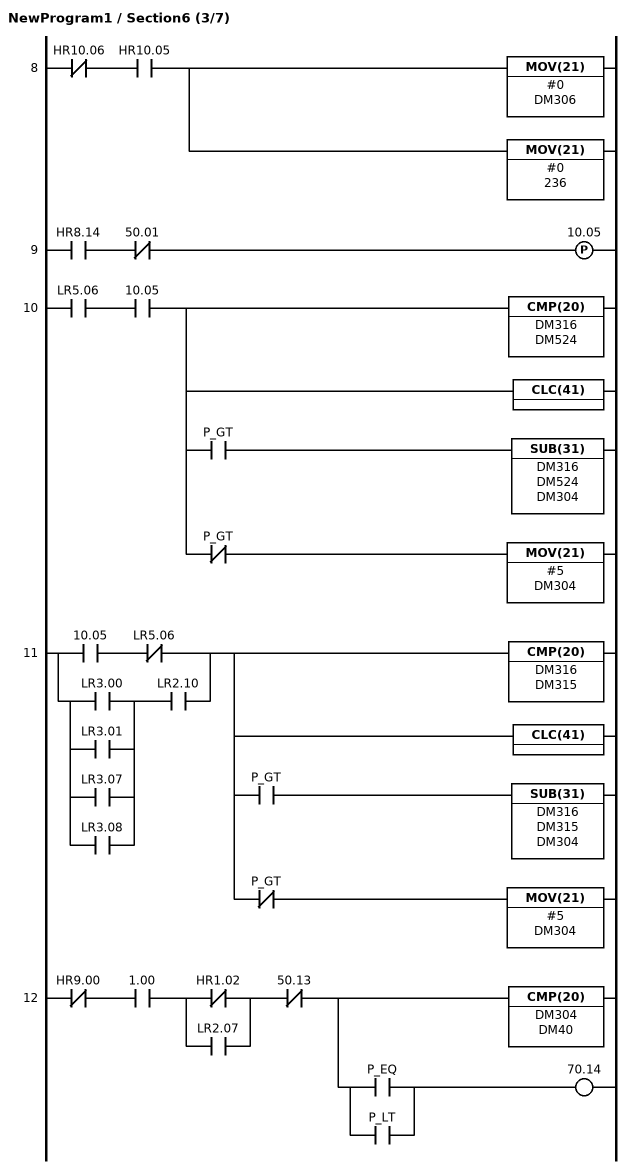
; [picture p48: NewProgram1 / Section6, rungs 8-12]
; rung 8
LDNOT HR10.06
AND HR10.05
MOV(21) #0 DM306
MOV(21) #0 236
; rung 9
LD HR8.14
ANDNOT 50.01
DIFU(13) 10.05
; rung 10
LD LR5.06
AND 10.05
OUT TR0
CMP(20) DM316 DM524
CLC(41)
AND P_GT
SUB(31) DM316 DM524 DM304
LD TR0
ANDNOT P_GT
MOV(21) #5 DM304
; rung 11
LD 10.05
ANDNOT LR5.06
LD LR3.00
OR LR3.01
OR LR3.07
OR LR3.08
AND LR2.10
ORLD
OUT TR0
CMP(20) DM316 DM315
CLC(41)
AND P_GT
SUB(31) DM316 DM315 DM304
LD TR0
ANDNOT P_GT
MOV(21) #5 DM304
; rung 12
LDNOT HR9.00
AND 1.00
LDNOT HR1.02
OR LR2.07
ANDLD
ANDNOT 50.13
CMP(20) DM304 DM40
LD P_EQ
OR P_LT
ANDLD
OUT 70.14

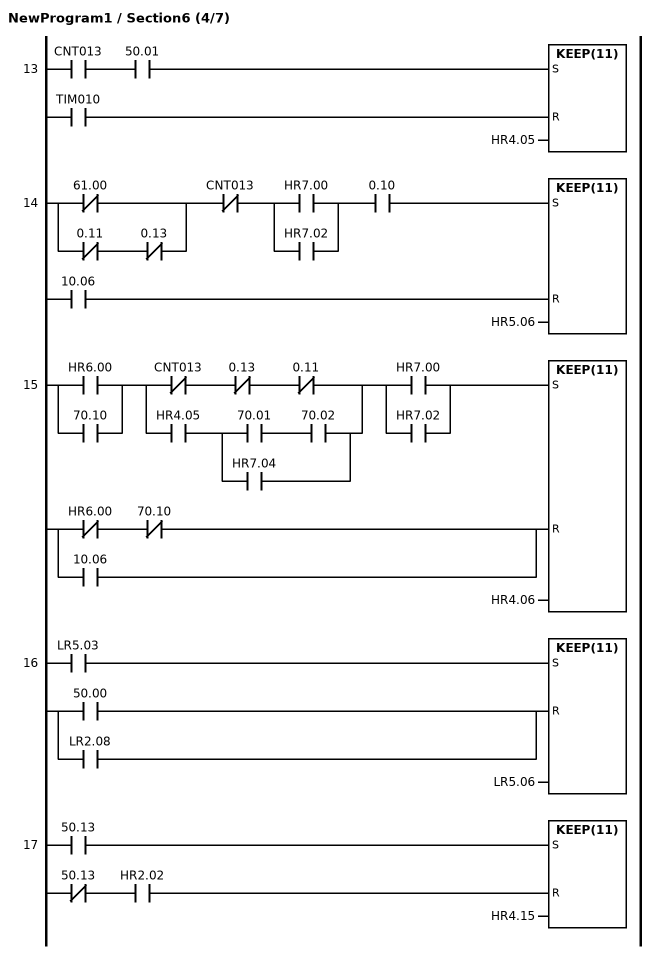
; rung 13
LD CNT013
AND 50.01
LD TIM010
KEEP(11) HR4.05
; rung 14
LDNOT 61.00
LDNOT 0.11
ANDNOT 0.13
ORLD
ANDNOT CNT013
LD HR7.00
OR HR7.02
ANDLD
AND 0.10
LD 10.06
KEEP(11) HR5.06
; rung 15
LD HR6.00
OR 70.10
LDNOT CNT013
ANDNOT 0.13
ANDNOT 0.11
LD HR4.05
LD 70.01
AND 70.02
OR HR7.04
ANDLD
ORLD
ANDLD
LD HR7.00
OR HR7.02
ANDLD
LDNOT HR6.00
ANDNOT 70.10
OR 10.06
KEEP(11) HR4.06
; rung 16
LD LR5.03
LD 50.00
OR LR2.08
KEEP(11) LR5.06
; rung 17
LD 50.13
LDNOT 50.13
AND HR2.02
KEEP(11) HR4.15

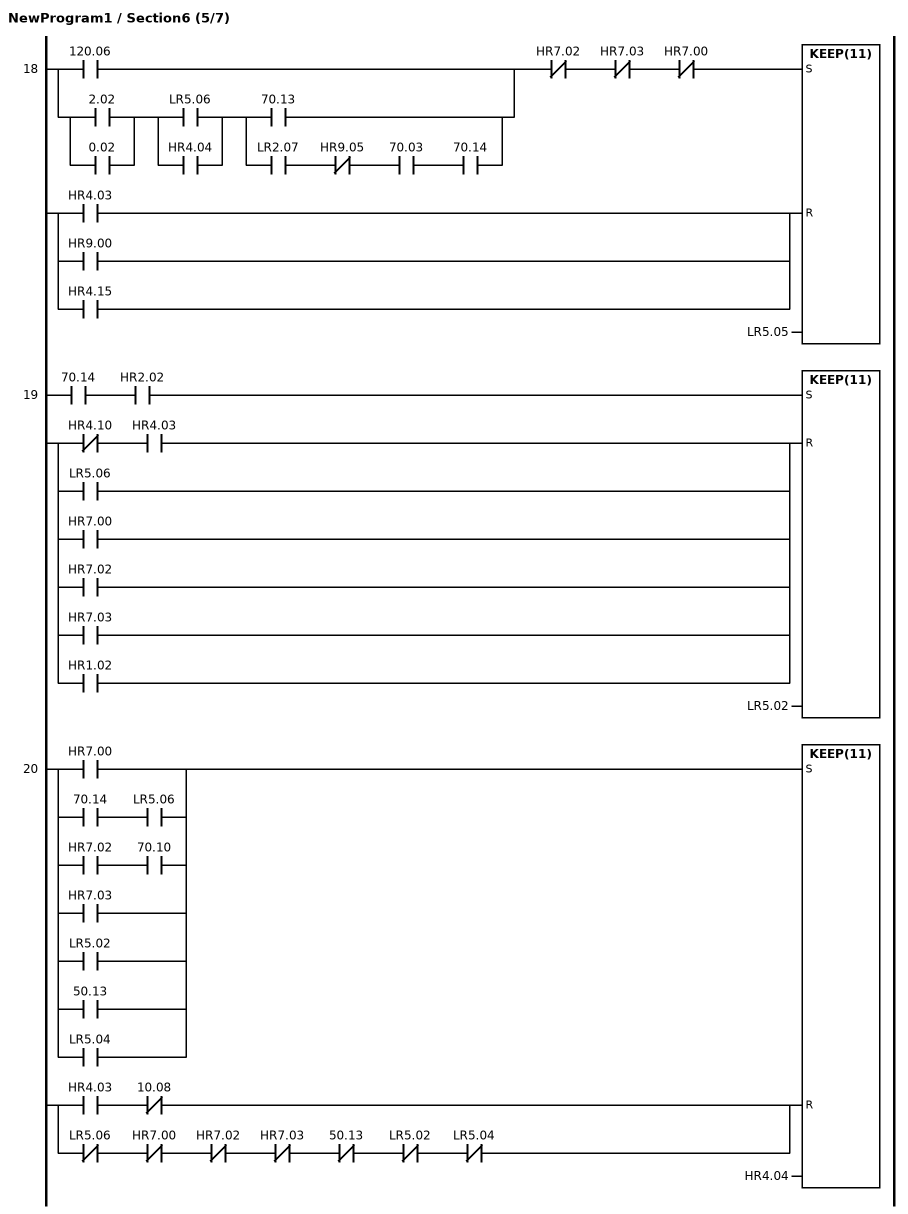
; rung 18
LD 120.06
LD 2.02
OR 0.02
LD LR5.06
OR HR4.04
ANDLD
LD 70.13
LD LR2.07
ANDNOT HR9.05
AND 70.03
AND 70.14
ORLD
ANDLD
ORLD
ANDNOT HR7.02
ANDNOT HR7.03
ANDNOT HR7.00
LD HR4.03
OR HR9.00
OR HR4.15
KEEP(11) LR5.05
; rung 19
LD 70.14
AND HR2.02
LDNOT HR4.10
AND HR4.03
OR LR5.06
OR HR7.00
OR HR7.02
OR HR7.03
OR HR1.02
KEEP(11) LR5.02
; rung 20
LD HR7.00
LD 70.14
AND LR5.06
ORLD
LD HR7.02
AND 70.10
ORLD
OR HR7.03
OR LR5.02
OR 50.13
OR LR5.04
LD HR4.03
ANDNOT 10.08
LDNOT LR5.06
ANDNOT HR7.00
ANDNOT HR7.02
ANDNOT HR7.03
ANDNOT 50.13
ANDNOT LR5.02
ANDNOT LR5.04
ORLD
KEEP(11) HR4.04

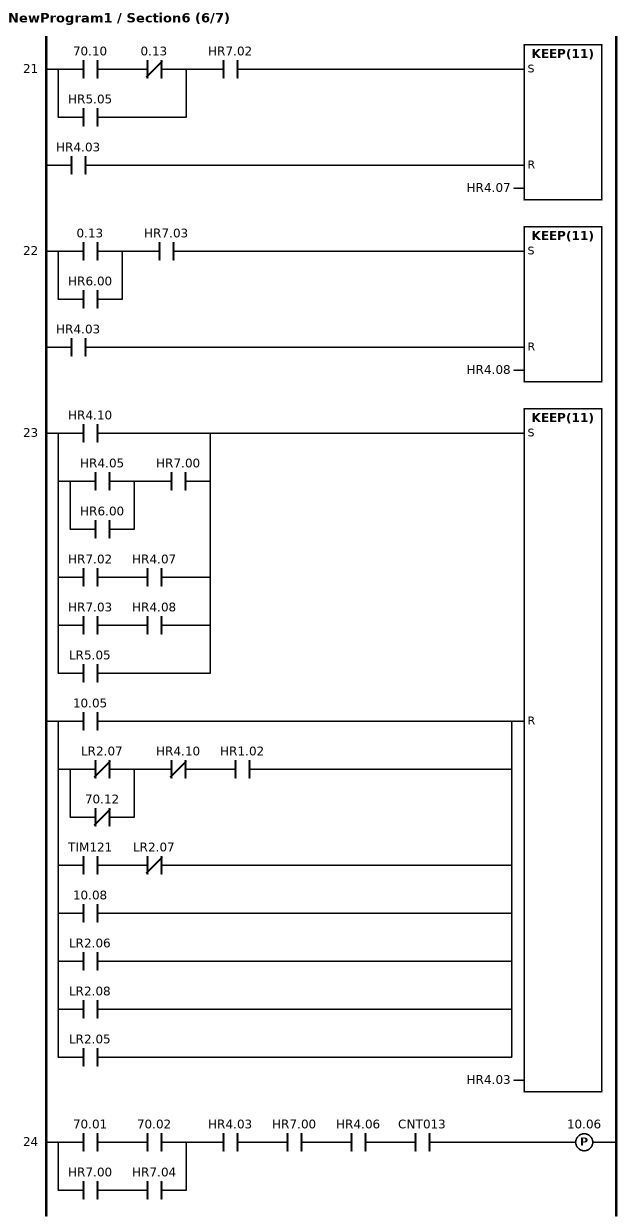
; rung 21
LD 70.10
ANDNOT 0.13
OR HR5.05
AND HR7.02
LD HR4.03
KEEP(11) HR4.07
; rung 22
LD 0.13
OR HR6.00
AND HR7.03
LD HR4.03
KEEP(11) HR4.08
; rung 23
LD HR4.10
LD HR4.05
OR HR6.00
AND HR7.00
ORLD
LD HR7.02
AND HR4.07
ORLD
LD HR7.03
AND HR4.08
ORLD
OR LR5.05
LD 10.05
LDNOT LR2.07
ORNOT 70.12
ANDNOT HR4.10
AND HR1.02
ORLD
LD TIM121
ANDNOT LR2.07
ORLD
OR 10.08
OR LR2.06
OR LR2.08
OR LR2.05
KEEP(11) HR4.03
; rung 24
LD 70.01
AND 70.02
LD HR7.00
AND HR7.04
ORLD
AND HR4.03
AND HR7.00
AND HR4.06
AND CNT013
DIFU(13) 10.06

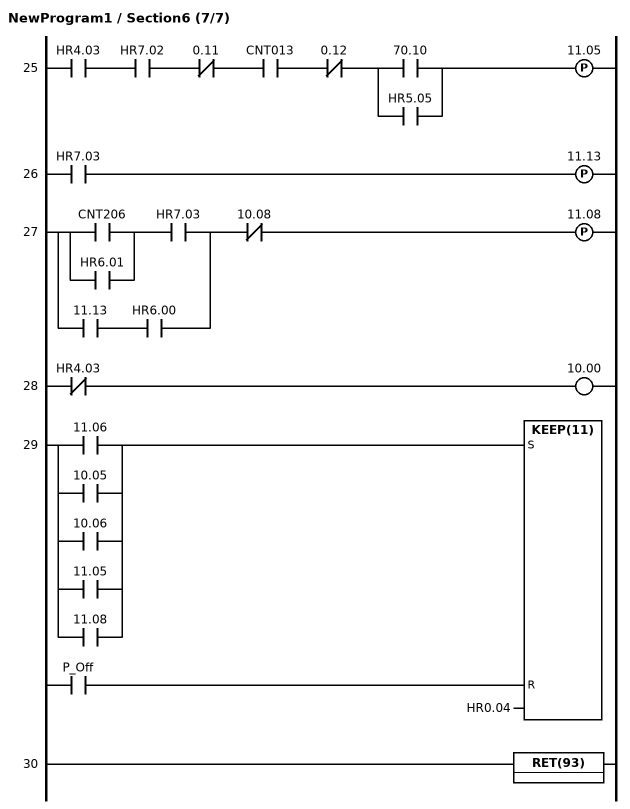
; rung 25
LD HR4.03
AND HR7.02
ANDNOT 0.11
AND CNT013
ANDNOT 0.12
LD 70.10
OR HR5.05
ANDLD
DIFU(13) 11.05
; rung 26
LD HR7.03
DIFU(13) 11.13
; rung 27
LD CNT206
OR HR6.01
AND HR7.03
LD 11.13
AND HR6.00
ORLD
ANDNOT 10.08
DIFU(13) 11.08
; rung 28
LDNOT HR4.03
OUT 10.00
; rung 29
LD 11.06
OR 10.05
OR 10.06
OR 11.05
OR 11.08
LD P_Off
KEEP(11) HR0.04
; rung 30
RET(93)

### Section Section7

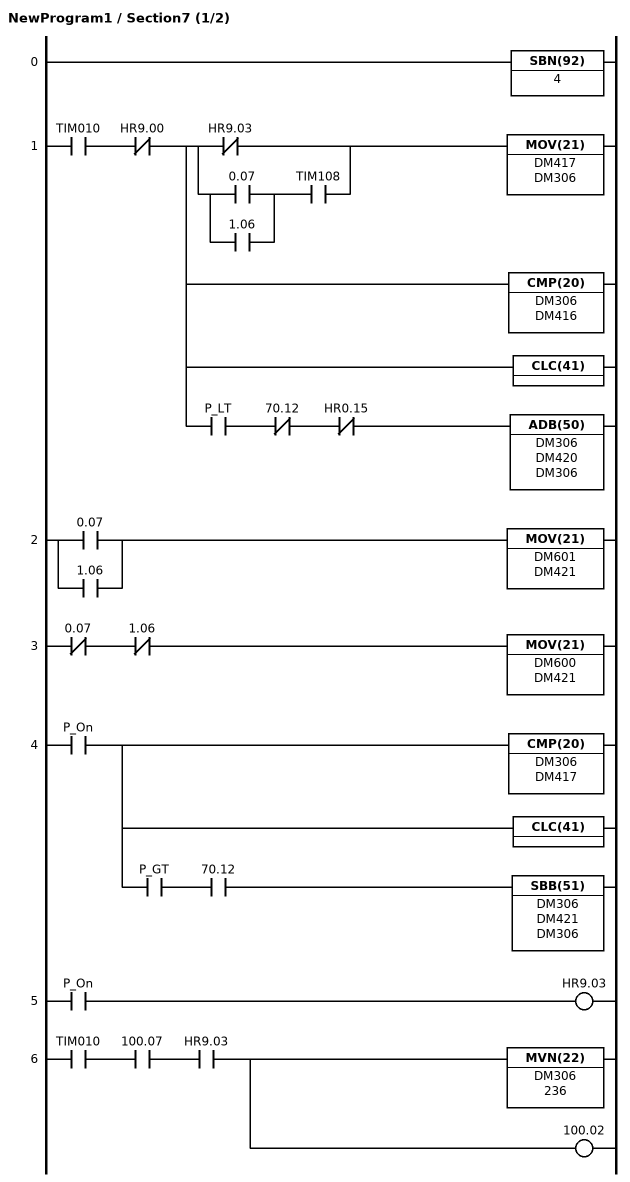
; rung 0
SBN(92) 4
; rung 1
LD TIM010
ANDNOT HR9.00
OUT TR0
LDNOT HR9.03
LD 0.07
OR 1.06
AND TIM108
ORLD
ANDLD
MOV(21) DM417 DM306
LD TR0
CMP(20) DM306 DM416
CLC(41)
AND P_LT
ANDNOT 70.12
ANDNOT HR0.15
ADB(50) DM306 DM420 DM306
; rung 2
LD 0.07
OR 1.06
MOV(21) DM601 DM421
; rung 3
LDNOT 0.07
ANDNOT 1.06
MOV(21) DM600 DM421
; rung 4
LD P_On
CMP(20) DM306 DM417
CLC(41)
AND P_GT
AND 70.12
SBB(51) DM306 DM421 DM306
; rung 5
LD P_On
OUT HR9.03
; rung 6
LD TIM010
AND 100.07
AND HR9.03
MVN(22) DM306 236
OUT 100.02

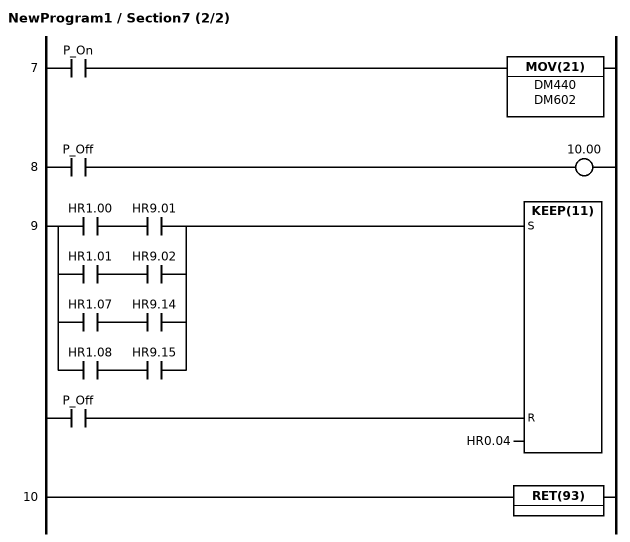
; rung 7
LD P_On
MOV(21) DM440 DM602
; rung 8
LD P_Off
OUT 10.00
; rung 9
LD HR1.00
AND HR9.01
LD HR1.01
AND HR9.02
ORLD
LD HR1.07
AND HR9.14
ORLD
LD HR1.08
AND HR9.15
ORLD
LD P_Off
KEEP(11) HR0.04
; rung 10
RET(93)

### Section Section8

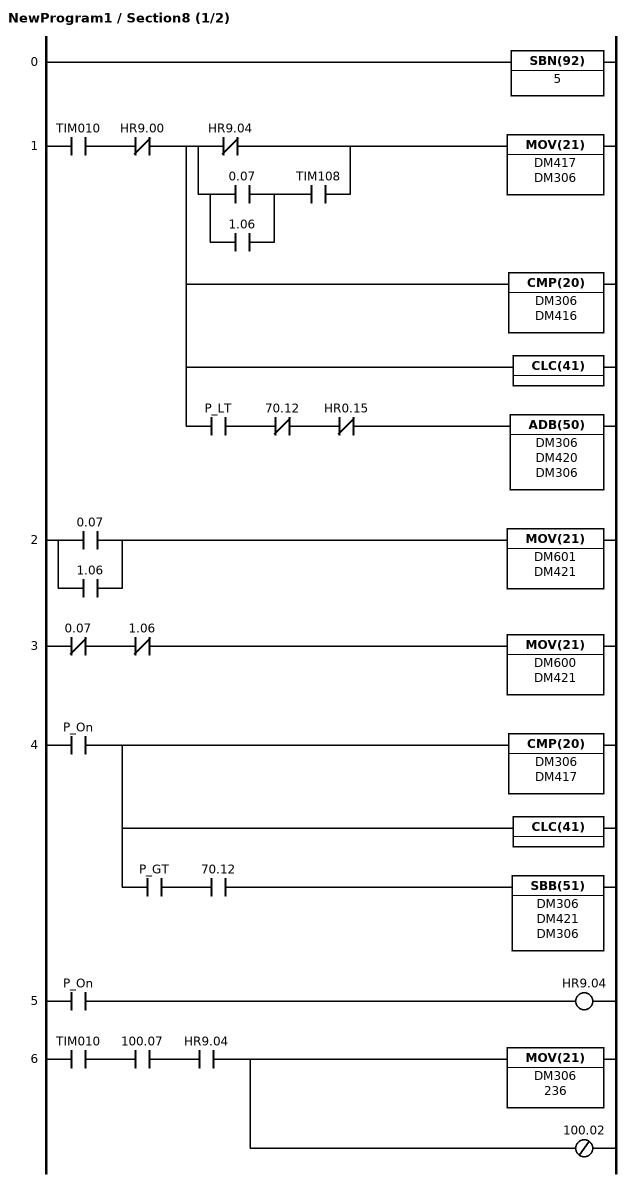
; rung 0
SBN(92) 5
; rung 1
LD TIM010
ANDNOT HR9.00
OUT TR0
LDNOT HR9.04
LD 0.07
OR 1.06
AND TIM108
ORLD
ANDLD
MOV(21) DM417 DM306
LD TR0
CMP(20) DM306 DM416
CLC(41)
AND P_LT
ANDNOT 70.12
ANDNOT HR0.15
ADB(50) DM306 DM420 DM306
; rung 2
LD 0.07
OR 1.06
MOV(21) DM601 DM421
; rung 3
LDNOT 0.07
ANDNOT 1.06
MOV(21) DM600 DM421
; rung 4
LD P_On
CMP(20) DM306 DM417
CLC(41)
AND P_GT
AND 70.12
SBB(51) DM306 DM421 DM306
; rung 5
LD P_On
OUT HR9.04
; rung 6
LD TIM010
AND 100.07
AND HR9.04
MOV(21) DM306 236
OUTNOT 100.02

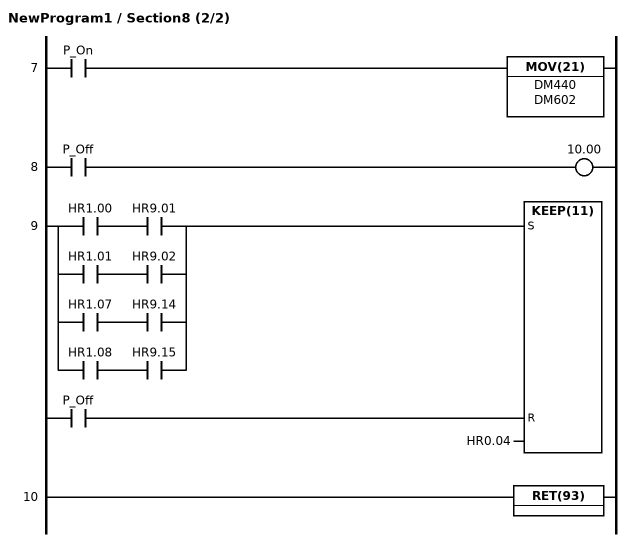
; rung 7
LD P_On
MOV(21) DM440 DM602
; rung 8
LD P_Off
OUT 10.00
; rung 9
LD HR1.00
AND HR9.01
LD HR1.01
AND HR9.02
ORLD
LD HR1.07
AND HR9.14
ORLD
LD HR1.08
AND HR9.15
ORLD
LD P_Off
KEEP(11) HR0.04
; rung 10
RET(93)

### Section Section9

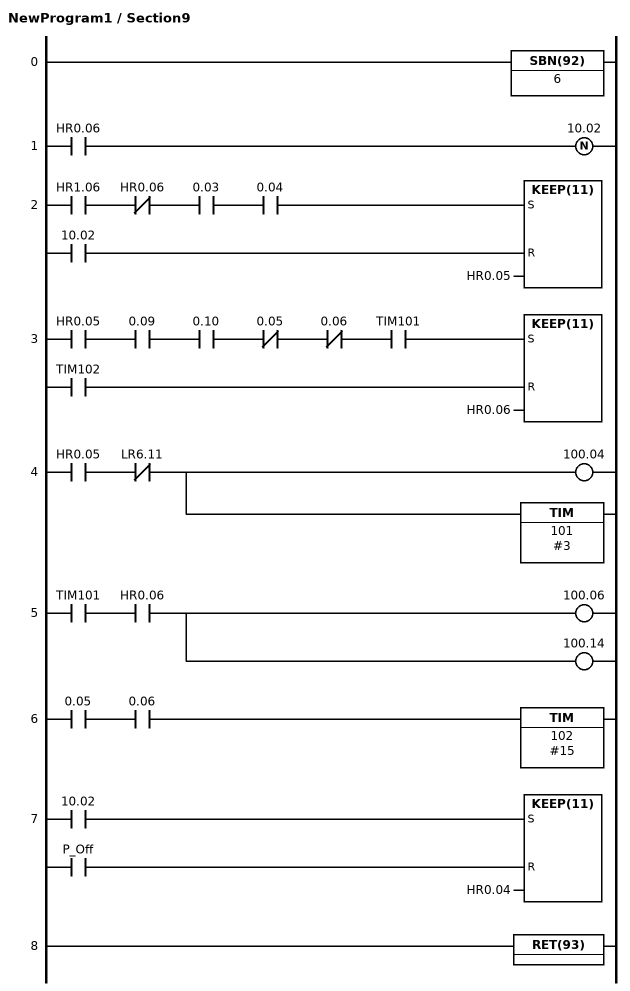
; rung 0
SBN(92) 6
; rung 1
LD HR0.06
DIFD(14) 10.02
; rung 2
LD HR1.06
ANDNOT HR0.06
AND 0.03
AND 0.04
LD 10.02
KEEP(11) HR0.05
; rung 3
LD HR0.05
AND 0.09
AND 0.10
ANDNOT 0.05
ANDNOT 0.06
AND TIM101
LD TIM102
KEEP(11) HR0.06
; rung 4
LD HR0.05
ANDNOT LR6.11
OUT 100.04
TIM 101 #3
; rung 5
LD TIM101
AND HR0.06
OUT 100.06
OUT 100.14
; rung 6
LD 0.05
AND 0.06
TIM 102 #15
; rung 7
LD 10.02
LD P_Off
KEEP(11) HR0.04
; rung 8
RET(93)

### Section Section10

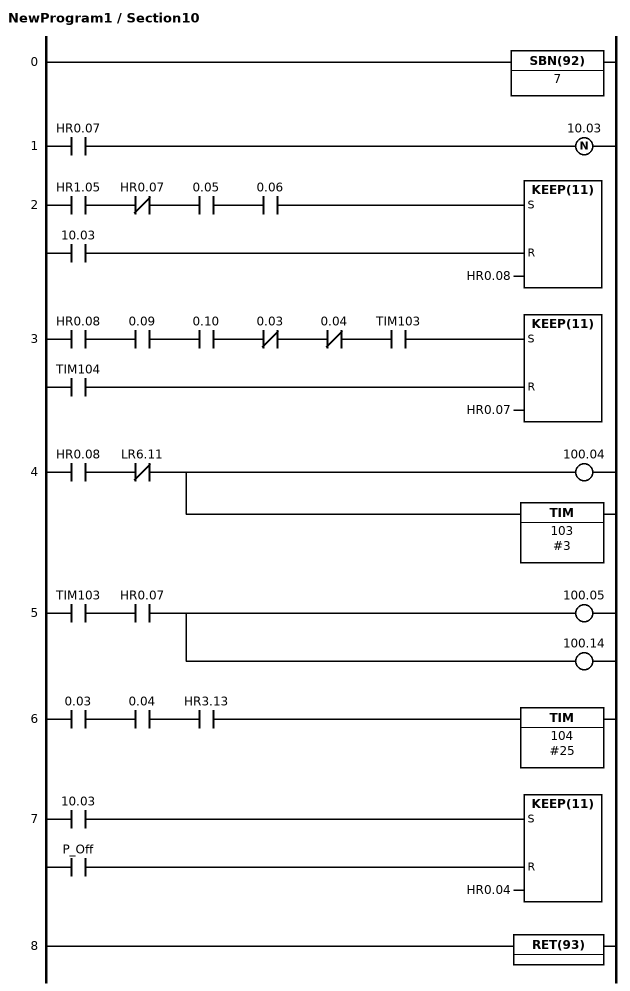
; rung 0
SBN(92) 7
; rung 1
LD HR0.07
DIFD(14) 10.03
; rung 2
LD HR1.05
ANDNOT HR0.07
AND 0.05
AND 0.06
LD 10.03
KEEP(11) HR0.08
; rung 3
LD HR0.08
AND 0.09
AND 0.10
ANDNOT 0.03
ANDNOT 0.04
AND TIM103
LD TIM104
KEEP(11) HR0.07
; rung 4
LD HR0.08
ANDNOT LR6.11
OUT 100.04
TIM 103 #3
; rung 5
LD TIM103
AND HR0.07
OUT 100.05
OUT 100.14
; rung 6
LD 0.03
AND 0.04
AND HR3.13
TIM 104 #25
; rung 7
LD 10.03
LD P_Off
KEEP(11) HR0.04
; rung 8
RET(93)

### Section Section11

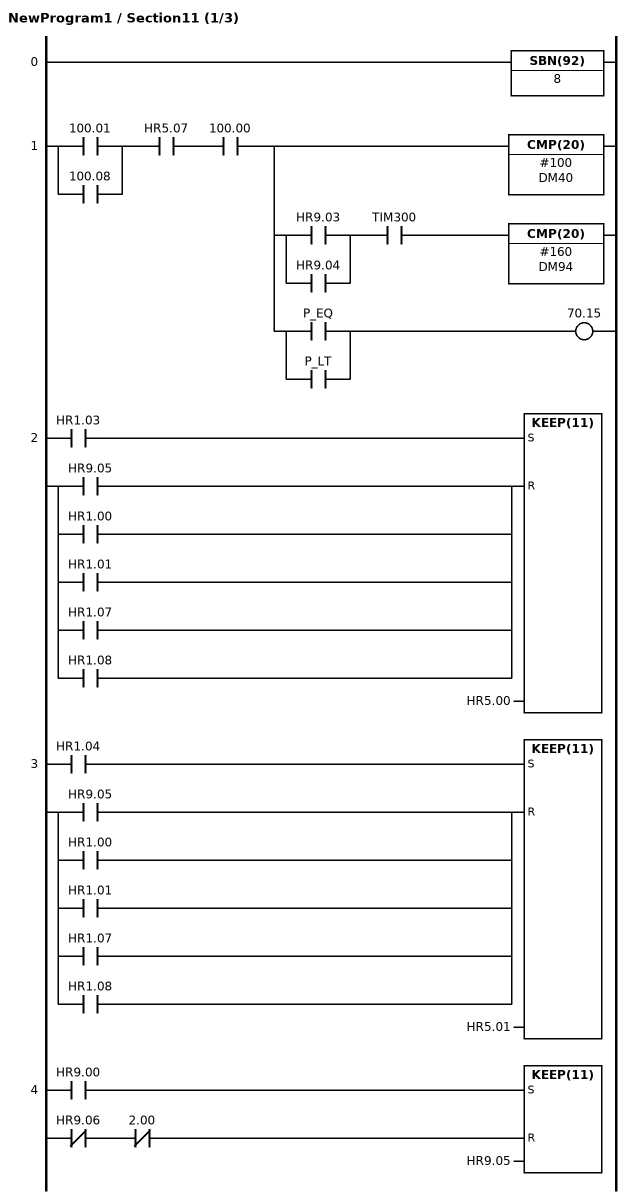
; rung 0
SBN(92) 8
; rung 1
LD 100.01
OR 100.08
AND HR5.07
AND 100.00
OUT TR0
CMP(20) #100 DM40
LD HR9.03
OR HR9.04
ANDLD
AND TIM300
CMP(20) #160 DM94
LD TR0
LD P_EQ
OR P_LT
ANDLD
OUT 70.15
; rung 2
LD HR1.03
LD HR9.05
OR HR1.00
OR HR1.01
OR HR1.07
OR HR1.08
KEEP(11) HR5.00
; rung 3
LD HR1.04
LD HR9.05
OR HR1.00
OR HR1.01
OR HR1.07
OR HR1.08
KEEP(11) HR5.01
; rung 4
LD HR9.00
LDNOT HR9.06
ANDNOT 2.00
KEEP(11) HR9.05

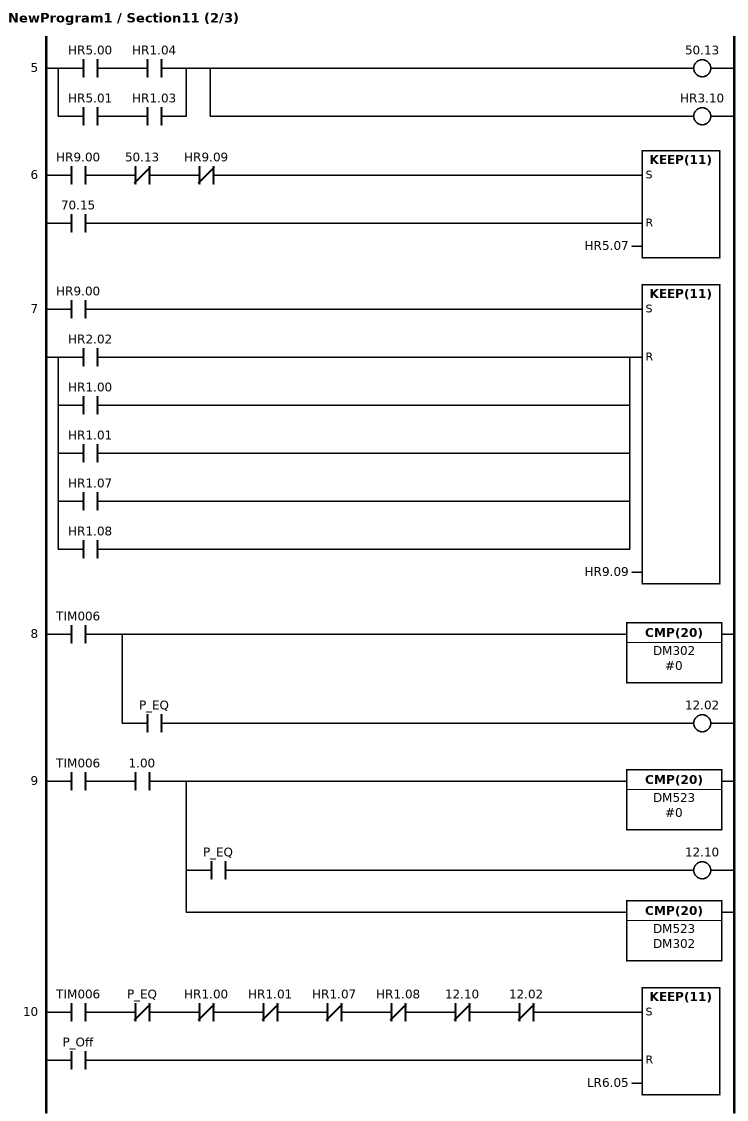
; rung 5
LD HR5.00
AND HR1.04
LD HR5.01
AND HR1.03
ORLD
OUT 50.13
OUT HR3.10
; rung 6
LD HR9.00
ANDNOT 50.13
ANDNOT HR9.09
LD 70.15
KEEP(11) HR5.07
; rung 7
LD HR9.00
LD HR2.02
OR HR1.00
OR HR1.01
OR HR1.07
OR HR1.08
KEEP(11) HR9.09
; rung 8
LD TIM006
CMP(20) DM302 #0
AND P_EQ
OUT 12.02
; rung 9
LD TIM006
AND 1.00
OUT TR0
CMP(20) DM523 #0
AND P_EQ
OUT 12.10
LD TR0
CMP(20) DM523 DM302
; rung 10
LD TIM006
ANDNOT P_EQ
ANDNOT HR1.00
ANDNOT HR1.01
ANDNOT HR1.07
ANDNOT HR1.08
ANDNOT 12.10
ANDNOT 12.02
LD P_Off
KEEP(11) LR6.05

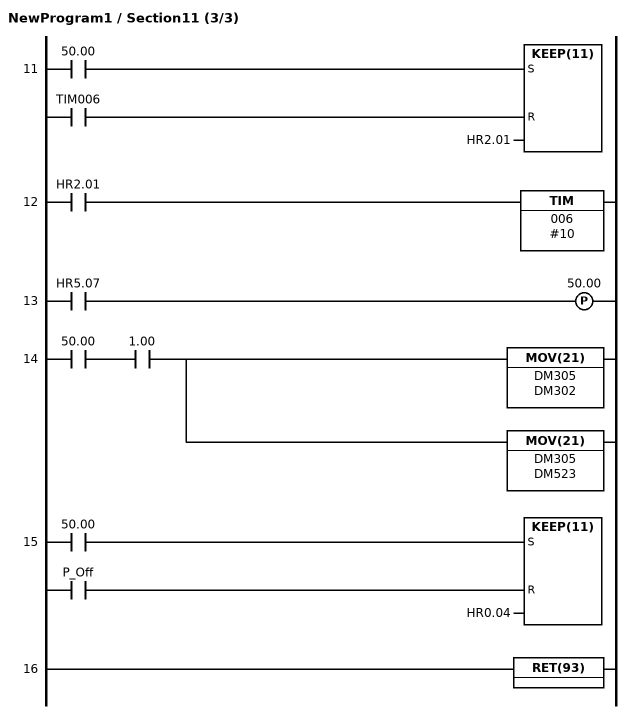
; rung 11
LD 50.00
LD TIM006
KEEP(11) HR2.01
; rung 12
LD HR2.01
TIM 006 #10
; rung 13
LD HR5.07
DIFU(13) 50.00
; rung 14
LD 50.00
AND 1.00
MOV(21) DM305 DM302
MOV(21) DM305 DM523
; rung 15
LD 50.00
LD P_Off
KEEP(11) HR0.04
; rung 16
RET(93)

### Section Section12

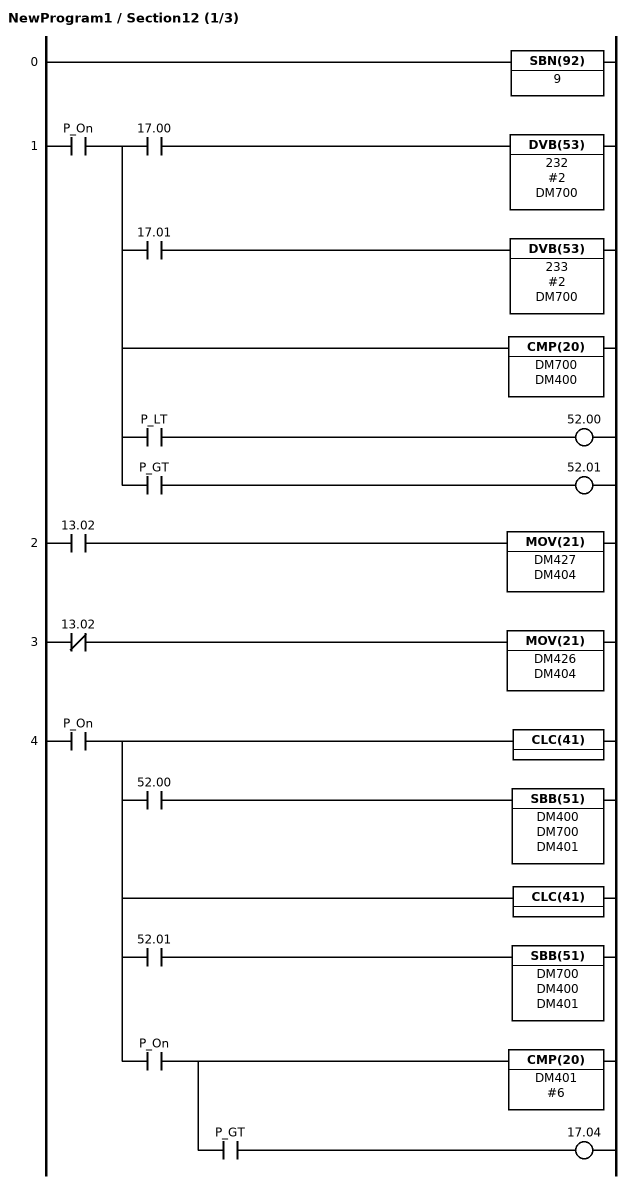
; rung 0
SBN(92) 9
; rung 1
LD P_On
OUT TR0
AND 17.00
DVB(53) 232 #2 DM700
LD TR0
AND 17.01
DVB(53) 233 #2 DM700
LD TR0
CMP(20) DM700 DM400
AND P_LT
OUT 52.00
LD TR0
AND P_GT
OUT 52.01
; rung 2
LD 13.02
MOV(21) DM427 DM404
; rung 3
LDNOT 13.02
MOV(21) DM426 DM404
; rung 4
LD P_On
OUT TR0
CLC(41)
AND 52.00
SBB(51) DM400 DM700 DM401
LD TR0
CLC(41)
AND 52.01
SBB(51) DM700 DM400 DM401
LD TR0
AND P_On
CMP(20) DM401 #6
AND P_GT
OUT 17.04

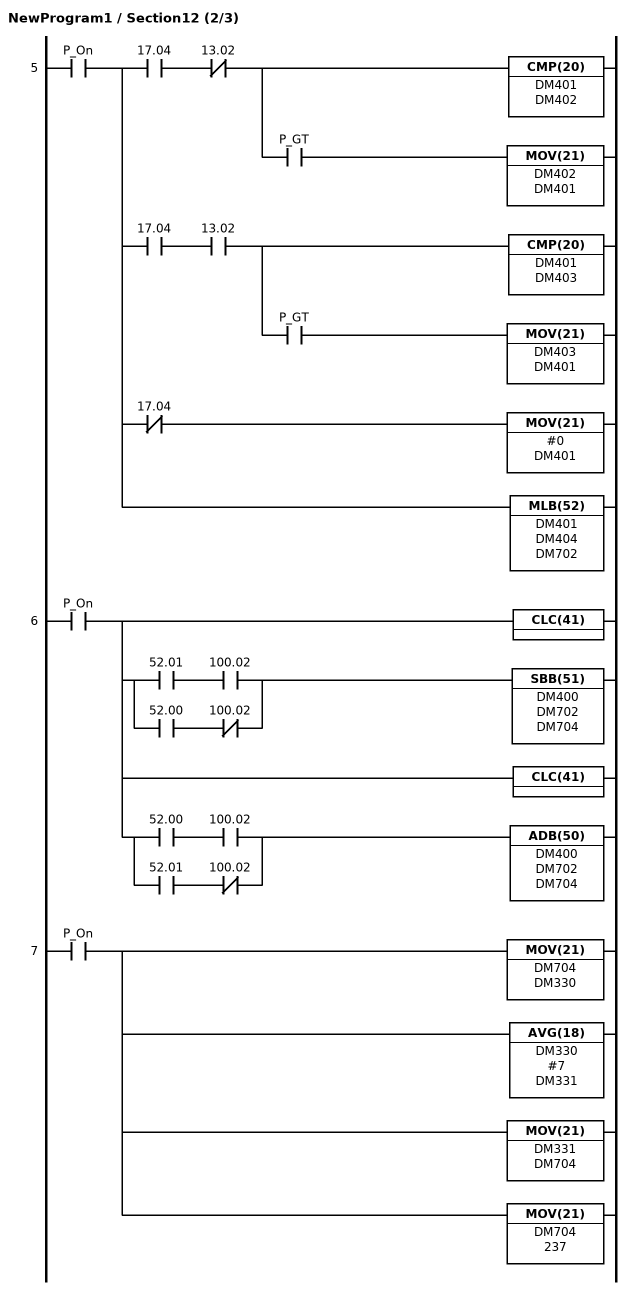
; rung 5
LD P_On
OUT TR0
AND 17.04
ANDNOT 13.02
CMP(20) DM401 DM402
AND P_GT
MOV(21) DM402 DM401
LD TR0
AND 17.04
AND 13.02
CMP(20) DM401 DM403
AND P_GT
MOV(21) DM403 DM401
LD TR0
ANDNOT 17.04
MOV(21) #0 DM401
LD TR0
MLB(52) DM401 DM404 DM702
; rung 6
LD P_On
OUT TR0
CLC(41)
LD 52.01
AND 100.02
LD 52.00
ANDNOT 100.02
ORLD
ANDLD
SBB(51) DM400 DM702 DM704
LD TR0
CLC(41)
LD 52.00
AND 100.02
LD 52.01
ANDNOT 100.02
ORLD
ANDLD
ADB(50) DM400 DM702 DM704
; rung 7
LD P_On
MOV(21) DM704 DM330
AVG(18) DM330 #7 DM331
MOV(21) DM331 DM704
MOV(21) DM704 237

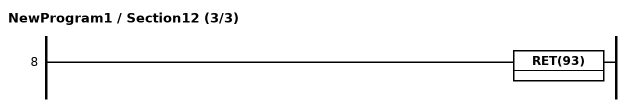
; rung 8
RET(93)

### Section Section13

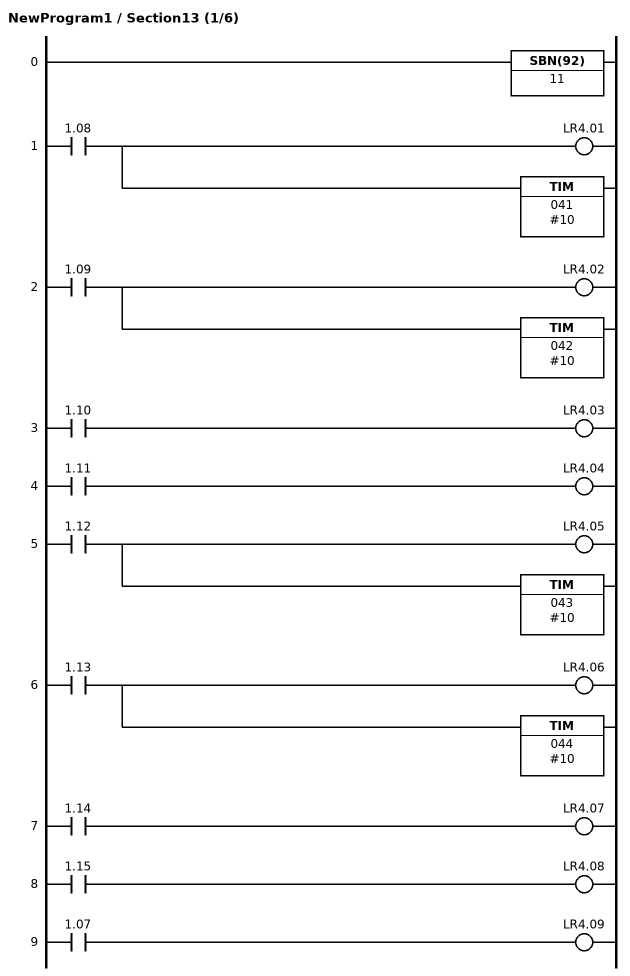
; rung 0
SBN(92) 11
; rung 1
LD 1.08
OUT LR4.01
TIM 041 #10
; rung 2
LD 1.09
OUT LR4.02
TIM 042 #10
; rung 3
LD 1.10
OUT LR4.03
; rung 4
LD 1.11
OUT LR4.04
; rung 5
LD 1.12
OUT LR4.05
TIM 043 #10
; rung 6
LD 1.13
OUT LR4.06
TIM 044 #10
; rung 7
LD 1.14
OUT LR4.07
; rung 8
LD 1.15
OUT LR4.08
; rung 9
LD 1.07
OUT LR4.09

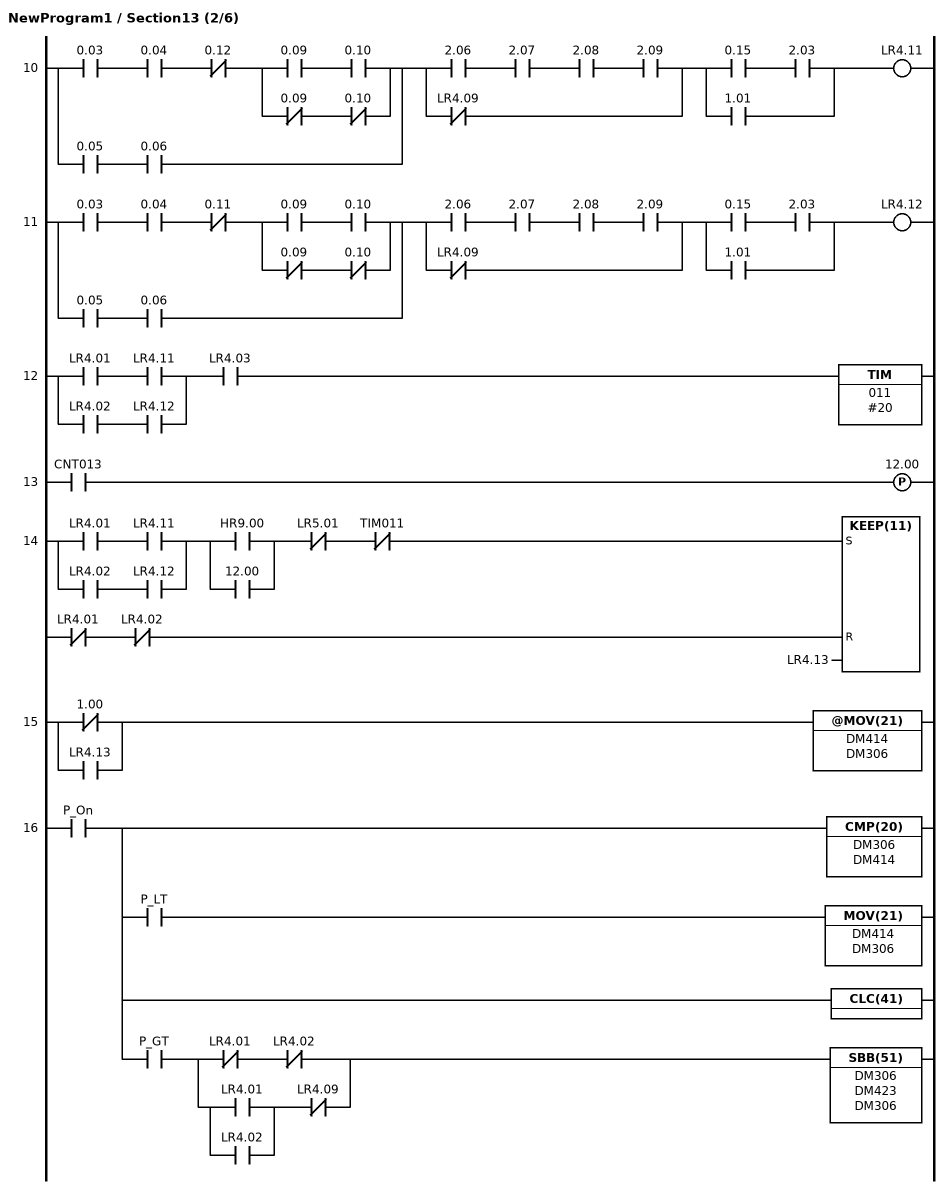
; rung 10
LD 0.03
AND 0.04
ANDNOT 0.12
LD 0.09
AND 0.10
LDNOT 0.09
ANDNOT 0.10
ORLD
ANDLD
LD 0.05
AND 0.06
ORLD
LD 2.06
AND 2.07
AND 2.08
AND 2.09
ORNOT LR4.09
ANDLD
LD 0.15
AND 2.03
OR 1.01
ANDLD
OUT LR4.11
; rung 11
LD 0.03
AND 0.04
ANDNOT 0.11
LD 0.09
AND 0.10
LDNOT 0.09
ANDNOT 0.10
ORLD
ANDLD
LD 0.05
AND 0.06
ORLD
LD 2.06
AND 2.07
AND 2.08
AND 2.09
ORNOT LR4.09
ANDLD
LD 0.15
AND 2.03
OR 1.01
ANDLD
OUT LR4.12
; rung 12
LD LR4.01
AND LR4.11
LD LR4.02
AND LR4.12
ORLD
AND LR4.03
TIM 011 #20
; rung 13
LD CNT013
DIFU(13) 12.00
; rung 14
LD LR4.01
AND LR4.11
LD LR4.02
AND LR4.12
ORLD
LD HR9.00
OR 12.00
ANDLD
ANDNOT LR5.01
ANDNOT TIM011
LDNOT LR4.01
ANDNOT LR4.02
KEEP(11) LR4.13
; rung 15
LDNOT 1.00
OR LR4.13
@MOV(21) DM414 DM306
; rung 16
LD P_On
OUT TR0
CMP(20) DM306 DM414
AND P_LT
MOV(21) DM414 DM306
LD TR0
CLC(41)
AND P_GT
LDNOT LR4.01
ANDNOT LR4.02
LD LR4.01
OR LR4.02
ANDNOT LR4.09
ORLD
ANDLD
SBB(51) DM306 DM423 DM306

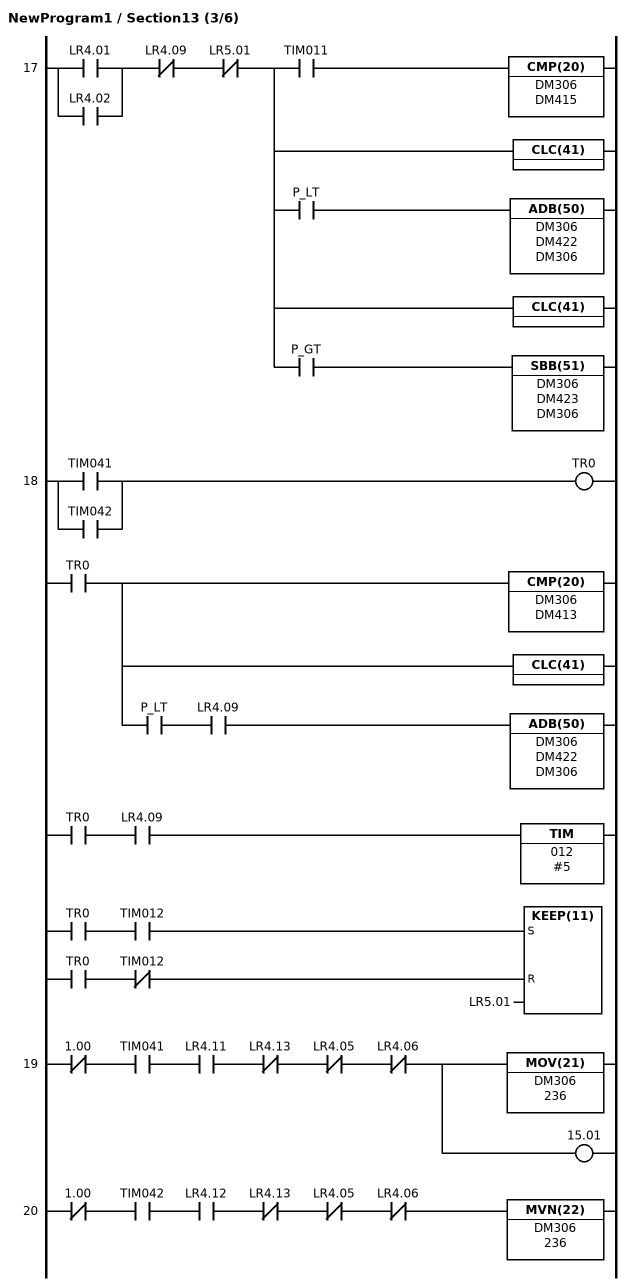
; rung 17
LD LR4.01
OR LR4.02
ANDNOT LR4.09
ANDNOT LR5.01
OUT TR0
AND TIM011
CMP(20) DM306 DM415
LD TR0
CLC(41)
AND P_LT
ADB(50) DM306 DM422 DM306
LD TR0
CLC(41)
AND P_GT
SBB(51) DM306 DM423 DM306
; rung 18
LD TIM041
OR TIM042
OUT TR0
CMP(20) DM306 DM413
CLC(41)
AND P_LT
AND LR4.09
ADB(50) DM306 DM422 DM306
LD TR0
AND LR4.09
TIM 012 #5
LD TR0
AND TIM012
LD TR0
ANDNOT TIM012
KEEP(11) LR5.01
; rung 19
LDNOT 1.00
AND TIM041
AND LR4.11
ANDNOT LR4.13
ANDNOT LR4.05
ANDNOT LR4.06
MOV(21) DM306 236
OUT 15.01
; rung 20
LDNOT 1.00
AND TIM042
AND LR4.12
ANDNOT LR4.13
ANDNOT LR4.05
ANDNOT LR4.06
MVN(22) DM306 236

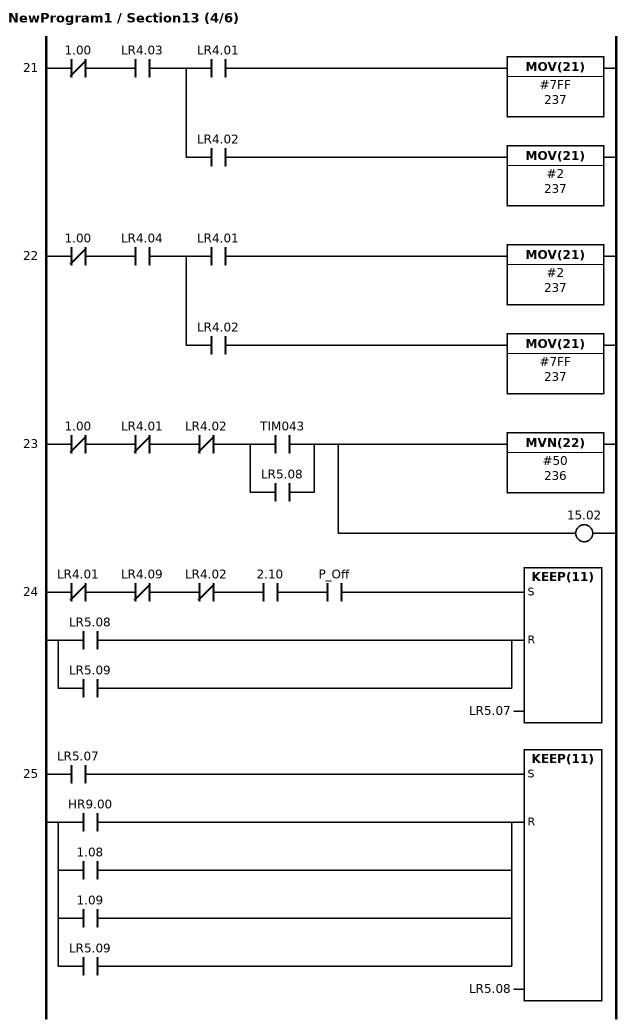
; rung 21
LDNOT 1.00
AND LR4.03
OUT TR0
AND LR4.01
MOV(21) #7FF 237
LD TR0
AND LR4.02
MOV(21) #2 237
; rung 22
LDNOT 1.00
AND LR4.04
OUT TR0
AND LR4.01
MOV(21) #2 237
LD TR0
AND LR4.02
MOV(21) #7FF 237
; rung 23
LDNOT 1.00
ANDNOT LR4.01
ANDNOT LR4.02
LD TIM043
OR LR5.08
ANDLD
MVN(22) #50 236
OUT 15.02
; rung 24
LDNOT LR4.01
ANDNOT LR4.09
ANDNOT LR4.02
AND 2.10
AND P_Off
LD LR5.08
OR LR5.09
KEEP(11) LR5.07
; rung 25
LD LR5.07
LD HR9.00
OR 1.08
OR 1.09
OR LR5.09
KEEP(11) LR5.08

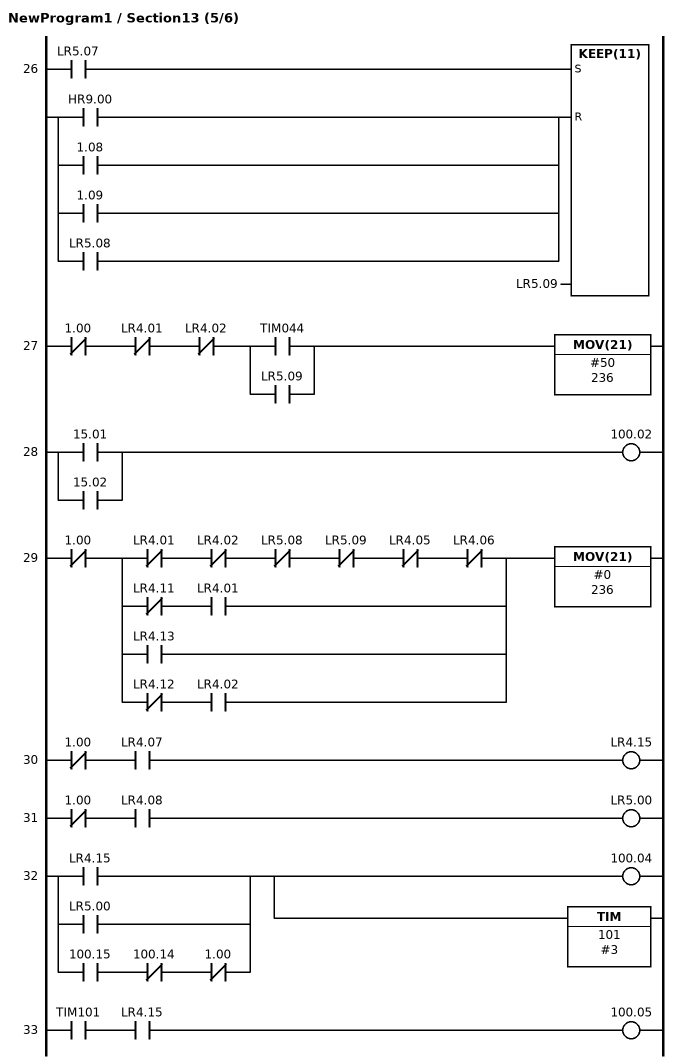
; rung 26
LD LR5.07
LD HR9.00
OR 1.08
OR 1.09
OR LR5.08
KEEP(11) LR5.09
; rung 27
LDNOT 1.00
ANDNOT LR4.01
ANDNOT LR4.02
LD TIM044
OR LR5.09
ANDLD
MOV(21) #50 236
; rung 28
LD 15.01
OR 15.02
OUT 100.02
; rung 29
LDNOT 1.00
LDNOT LR4.01
ANDNOT LR4.02
ANDNOT LR5.08
ANDNOT LR5.09
ANDNOT LR4.05
ANDNOT LR4.06
LDNOT LR4.11
AND LR4.01
ORLD
OR LR4.13
LDNOT LR4.12
AND LR4.02
ORLD
ANDLD
MOV(21) #0 236
; rung 30
LDNOT 1.00
AND LR4.07
OUT LR4.15
; rung 31
LDNOT 1.00
AND LR4.08
OUT LR5.00
; rung 32
LD LR4.15
OR LR5.00
LD 100.15
ANDNOT 100.14
ANDNOT 1.00
ORLD
OUT 100.04
TIM 101 #3
; rung 33
LD TIM101
AND LR4.15
OUT 100.05

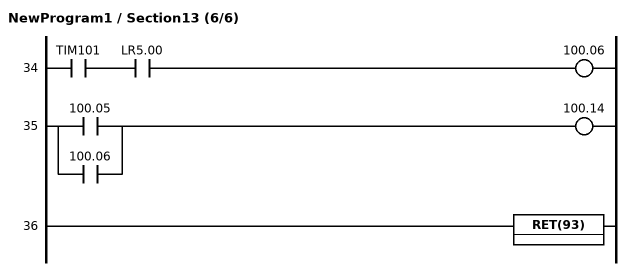
; rung 34
LD TIM101
AND LR5.00
OUT 100.06
; rung 35
LD 100.05
OR 100.06
OUT 100.14
; rung 36
RET(93)

### Section Section14

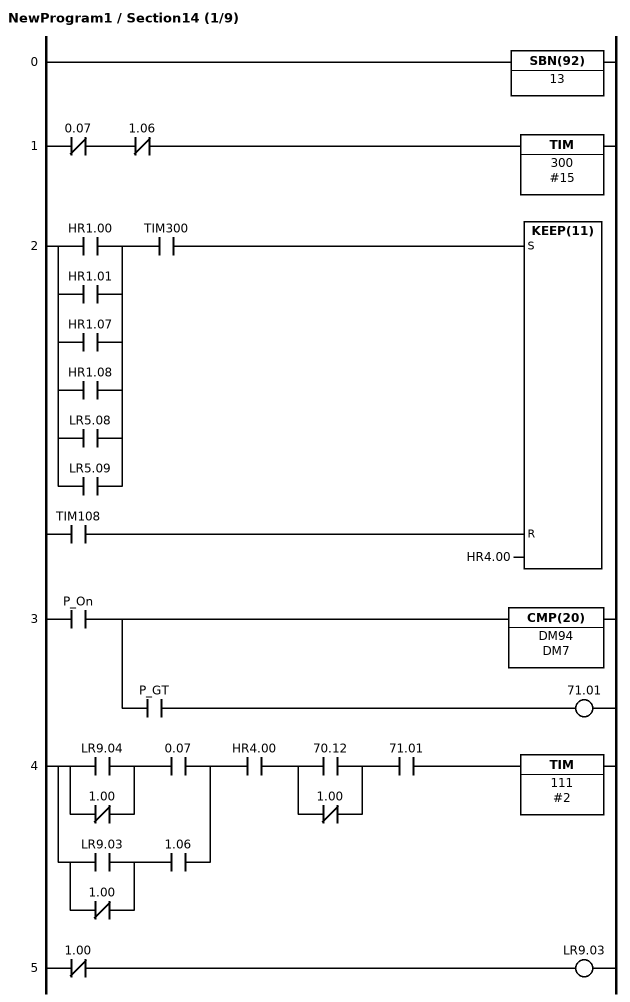
; rung 0
SBN(92) 13
; rung 1
LDNOT 0.07
ANDNOT 1.06
TIM 300 #15
; rung 2
LD HR1.00
OR HR1.01
OR HR1.07
OR HR1.08
OR LR5.08
OR LR5.09
AND TIM300
LD TIM108
KEEP(11) HR4.00
; rung 3
LD P_On
CMP(20) DM94 DM7
AND P_GT
OUT 71.01
; rung 4
LD LR9.04
ORNOT 1.00
AND 0.07
LD LR9.03
ORNOT 1.00
AND 1.06
ORLD
AND HR4.00
LD 70.12
ORNOT 1.00
ANDLD
AND 71.01
TIM 111 #2
; rung 5
LDNOT 1.00
OUT LR9.03

